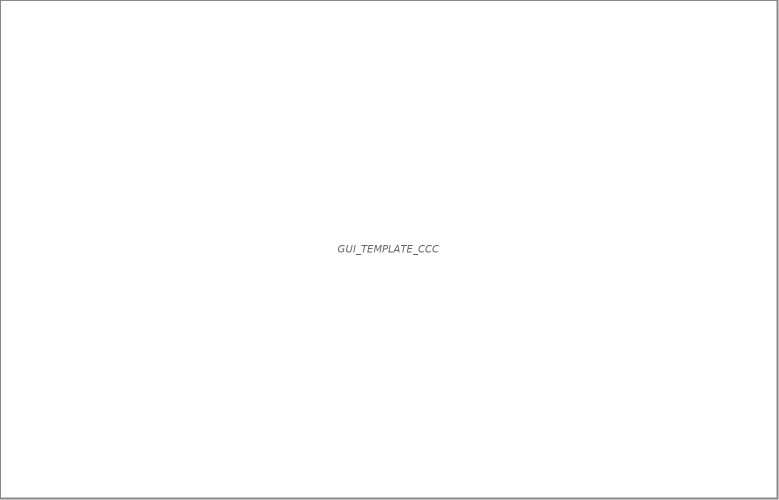
VISUALIZATION GUI_CCC  // 779x500
    Frame (0,0 777x498)
        shows GUI_TEMPLATE_CCC(m_Instance := MAIN.CCC)
END_VISUALIZATION

(* stored: Version 1.1.0.1, ProductVersion 3.1.4022.16
   Visu GUI_CCC: Id {8761305a-3140-4b60-96ab-09df7fe1bba0} *)
